TYPE DUT_HOMS :
STRUCT
	// System initializiation
	fbRunHOMS : FB_RunHOMS;

	// Couple/Decouple motors
	{attribute 'pytmc' := '
		pv: COUPLE_Y
		io: o
	'}
	bExecuteCoupleY : BOOL;
	{attribute 'pytmc' := '
		pv: DECOUPLE_Y
		io: o
	'}
	bExecuteDecoupleY : BOOL;
	{attribute 'pytmc' := '
		pv: COUPLE_X
		io: o
	'}
	bExecuteCoupleX : BOOL;
	{attribute 'pytmc' := '
		pv: DECOUPLE_X
		io: o
	'}
	bExecuteDecoupleX : BOOL;

	// Coupling status
	{attribute 'pytmc' := '
		pv: ALREADY_COUPLED_Y
		io: i
        field: ZSV MAJOR
	'}
	bGantryAlreadyCoupledY : BOOL;
	{attribute 'pytmc' := '
		pv: ALREADY_COUPLED_X
		io: i
        field: ZSV MAJOR
	'}
	bGantryAlreadyCoupledX : BOOL;

	// Current gantry differences
	nCurrGantryY : LINT; // encoder counts = nm
	nCurrGantryX : LINT; // encoder counts = nm

	// Convert gantry differences to um (smaller number) to readout in epics
	{attribute 'pytmc' := '
		pv: GANTRY_Y
		field: EGU um
		io: i
	'}
	fCurrGantryY_um : REAL; // Y Gantry difference in um
	{attribute 'pytmc' := '
		pv: GANTRY_X
		field: EGU um
		io: i
	'}
	fCurrGantryX_um : REAL; // X Gantry difference in um
END_STRUCT
END_TYPE

(* stored: Version 1.1.0.1, ProductVersion 3.1.4022.18
   DUT DUT_HOMS: Id {0a6ad08f-c6e6-47f2-ab1c-db91063eb2d4} *)
